FUNCTION CallHardwareModules : BOOL //only purpose of this function is to call modules from Hardware

robot3();
robot4();

skidA22Left(slots := skidHmiA22Left);
skidA22Right(slots := skidHmiA22Right);

magazineA22Left(slots := magazineHmiA22Left);
magazineA22Right(slots := magazineHmiA22Right);

wrapperA22();
benderA22Left();

horizontalDriveA22Left();
horizontalDriveA22Right();

verticalDriveA22Left();
verticalDriveA22Right();

pistonA22Bottom();

END_FUNCTION

(* stored: Version 1.1.0.1, ProductVersion 3.1.4024.11
   POU CallHardwareModules: Id {d53bfde7-ef31-4033-a59e-17a8585cdf25}, SpecialFunc None *)
